// TwinCAT 3 PLC project PLC1
// ProgramVersion: 3.1.4026.21
// libraries:
//   Tc2_Standard, * (Beckhoff Automation GmbH)
//   Tc2_System, * (Beckhoff Automation GmbH)
//   Tc3_Module, * (Beckhoff Automation GmbH)
// project tree:
//   DUTs/ Jog_FxA_Type.TcDUT, Jog_FxB_Type.TcDUT, LaserJog.TcDUT, LaserVar.TcDUT, MyCustomType.TcDUT, SideClampVar.TcDUT
//   GVLs/ GVL.TcGVL, GVL_Main.TcGVL, Hmi_web.TcGVL
//   / PlcTask.TcTTO
//   POUs/ MAIN.TcPOU
// real-time tasks:
//   TASK PlcTask: cycle T#10ms, priority 20, ADS port 350

CONFIGURATION PLC1
    RESOURCE PLC ON TwinCAT3
        TASK PlcTask(INTERVAL := T#10ms, PRIORITY := 20);
        PROGRAM MAIN WITH PlcTask : MAIN;
    END_RESOURCE
END_CONFIGURATION

// ---- DUTs/Jog_FxA_Type.TcDUT
TYPE Jog_FxA_Type :
STRUCT
	
 H_Open:  BOOL;
 H_Open_S:  BOOL;
 H_Close:  BOOL;
 H_Close_S:  BOOL;

 H_Hold:  BOOL;
 H_Hold_S:  BOOL;

 V_Open:  BOOL;
 V_Open_S: BOOL;
 V_Close: BOOL;
 V_Close_S: BOOL;
  P : BOOL;
 P_S : BOOL;
 N : BOOL;
 N_S : BOOL;
 P_Fast : BOOL;
 P_Fast_S : BOOL;
 N_Fast : BOOL;
 N_Fast_S : BOOL;
END_STRUCT
END_TYPE

// ---- DUTs/Jog_FxB_Type.TcDUT
TYPE Jog_FxB_Type :
STRUCT
	 H_Open:  BOOL;
 H_Open_S:  BOOL;
 H_Close:  BOOL;
 H_Close_S:  BOOL;

 H_Hold:  BOOL;
 H_Hold_S:  BOOL;

 V_Open:  BOOL;
 V_Open_S: BOOL;
 V_Close: BOOL;
 V_Close_S: BOOL;

 
END_STRUCT
END_TYPE

// ---- DUTs/LaserJog.TcDUT
TYPE LaserJog :
STRUCT
	 X_P: BOOL;
     X_N: BOOL;
     X_H: BOOL;
	 
	 
	 X_P_S: BOOL;
     X_N_S: BOOL;
     X_H_S: BOOL;
	 
     Y_P: BOOL;
     Y_N: BOOL;
     Y_H: BOOL;
	 
	 
     Y_P_S: BOOL;
     Y_N_S: BOOL;
     Y_H_S: BOOL;
	 
     Z_P: BOOL;
     Z_N: BOOL;
     Z_H: BOOL;
	 
     Z_P_S: BOOL;
     Z_N_S: BOOL;
     Z_H_S: BOOL;
     Laser_Preview:BOOL;
     Laser_Preview_Select: INT	;
     Laser_Blow: BOOL;
     Laser_Cover: BOOL;

END_STRUCT
END_TYPE

// ---- DUTs/LaserVar.TcDUT
TYPE LaserVar :
STRUCT
    sv_bPLCHandShaking : BOOL;
    sv_bIPCHandShaking    : BOOL;
END_STRUCT
END_TYPE

// ---- DUTs/MyCustomType.TcDUT
TYPE MyCustomType :
STRUCT
    isActive : BOOL;
    speed    : REAL;
    counter  : INT;
END_STRUCT
END_TYPE

// ---- DUTs/SideClampVar.TcDUT
TYPE SideClampVar :
STRUCT
    sv_bButtonFwd: BOOL;
	sv_bButtonBwd: BOOL;
END_STRUCT
END_TYPE

// ---- GVLs/GVL.TcGVL
{attribute 'qualified_only'}
VAR_GLOBAL
END_VAR

// ---- GVLs/GVL_Main.TcGVL
{attribute 'qualified_only'}
VAR_GLOBAL
    g_bStart     : BOOL := FALSE;
    g_iCounter   : INT := 0;
    g_fSpeed     : REAL := 1.5;
    testBoolean     : BOOL := FALSE;
	
 g_machineStatus : MyCustomType := (
        isActive := FALSE,
        speed    := 0.0,
        counter  := 0
    );
	

LaserVars1:LaserVar := (
sv_bPLCHandShaking:= FALSE,
sv_bIPCHandShaking:= FALSE
    );
	LaserVars2:LaserVar := (
sv_bPLCHandShaking:= FALSE,
sv_bIPCHandShaking:= FALSE
    );
	LaserVars3:LaserVar := (
sv_bPLCHandShaking:= FALSE,
sv_bIPCHandShaking:= FALSE
    );
	LaserVars4:LaserVar := (
sv_bPLCHandShaking:= FALSE,
sv_bIPCHandShaking:= FALSE
    );

	
SideClampVars1:SideClampVar := (
sv_bButtonFwd:= FALSE,
sv_bButtonBwd:= FALSE);
	
SideClampVars2:SideClampVar := (
sv_bButtonFwd:= FALSE,
sv_bButtonBwd:= FALSE
 );
	
	

	
	
	
	
	
	
	
	
END_VAR

// ---- GVLs/Hmi_web.TcGVL
{attribute 'qualified_only'}
VAR_GLOBAL
    Jog_Speed: INT;
 Oil_Pump:BOOL;
Jog_FxA:Jog_FxA_Type:= (
      H_Open:= FALSE,
      H_Open_S:= FALSE,
      H_Close:= FALSE,
      H_Close_S:= FALSE,

      H_Hold:= FALSE,
      H_Hold_S:= FALSE,

      V_Open:= FALSE,
      V_Open_S:= FALSE,
      V_Close:= FALSE,
      V_Close_S:= FALSE,
   
     P:= FALSE,
      P_S:= FALSE,
      N:= FALSE,
      N_S:= FALSE,
      P_Fast:= FALSE,
      P_Fast_S:= FALSE,
      N_Fast:= FALSE,
      N_Fast_S:= FALSE
    );
 
 
Jog_FxB : Jog_FxB_Type := (
       H_Open:= FALSE,
      H_Open_S:= FALSE,
      H_Close:= FALSE,
      H_Close_S:= FALSE,

      H_Hold:= FALSE,
      H_Hold_S:= FALSE,

      V_Open:= FALSE,
      V_Open_S:= FALSE,
      V_Close:= FALSE,
      V_Close_S:= FALSE

    
);


 

//右軸
Jog_Ga: LaserJog:=( 
     X_P:= FALSE,
     X_N:= FALSE,
     X_H:= FALSE,
     Y_P:= FALSE,
     Y_N:= FALSE,
     Y_H:= FALSE,
     Z_P:= FALSE,
     Z_N:= FALSE,
     Z_H:= FALSE,
     Laser_Preview:=FALSE,
     Laser_Preview_Select:= 1,
     Laser_Blow:= FALSE,
     Laser_Cover:= FALSE);
//上軸
    Jog_Gb: LaserJog:=( 
     X_P:= FALSE,
     X_N:= FALSE,
     X_H:= FALSE,
     Y_P:= FALSE,
     Y_N:= FALSE,
     Y_H:= FALSE,
     Z_P:= FALSE,
     Z_N:= FALSE,
     Z_H:= FALSE,
     Laser_Preview:=FALSE,
     Laser_Preview_Select:= 1,
     Laser_Blow:= FALSE,
     Laser_Cover:= FALSE);
//左軸
    Jog_Gc: LaserJog:=( 
     X_P:= FALSE,
     X_N:= FALSE,
     X_H:= FALSE,
     Y_P:= FALSE,
     Y_N:= FALSE,
     Y_H:= FALSE,
     Z_P:= FALSE,
     Z_N:= FALSE,
     Z_H:= FALSE,
     Laser_Preview:=FALSE,
     Laser_Preview_Select:= 1,
     Laser_Blow:= FALSE,
     Laser_Cover:= FALSE);
//下軸
    Jog_Gd: LaserJog:=( 
     X_P:= FALSE,
     X_N:= FALSE,
     X_H:= FALSE,
     Y_P:= FALSE,
     Y_N:= FALSE,
     Y_H:= FALSE,
     Z_P:= FALSE,
     Z_N:= FALSE,
     Z_H:= FALSE,
     Laser_Preview:=FALSE,
     Laser_Preview_Select:= 1,
     Laser_Blow:= FALSE,
     Laser_Cover:= FALSE);


 	//*自動加工 */
    Auto_Start:  BOOL;
    //插單*/
    Auto_OneCycle_Start:  BOOL;
 	// 自動流程 加工單
	Auto_ProjectWorkOrder_uuid: STRING;
	// 排版專案 
    Start_WorkOrder_UUID: STRING;
	// 加工data_uuid
    Process_Data_UUID: STRING;
	// 雷標動作啟動 
    Process_Data_UUID_Start: BOOL;
 
 
 

    //動力滾輪
    Roller_Fwd:  BOOL;
    Roller_Fwd_S:  BOOL;
    //動力滾輪反轉
    Roller_Rev:  BOOL;
    Roller_Rev_S:  BOOL;

    //滾輪上浮
    Roller_Up:  BOOL;
    Roller_Up_S:  BOOL;
    //滾輪下降
    Roller_Down:  BOOL;
    Roller_Down_S:  BOOL;

    //入口料架-出口料架(0/1)*/
    Site_Select:  INT;
    //料架速率(0/1)*/
    Speed_Select:  INT;

    // 指定橫移->用二進位儲存 */
    Module_Select:  INT;

    //料架動作-台車前進*/
    Car_Rev:  BOOL;
    Car_Rev_S:  BOOL;
    //料架動作-台車後退
    Car_Fwd:  BOOL;
    Car_Fwd_S:  BOOL;
    //料架動作-台車上升
    Car_Up: BOOL;
    Car_Up_S:  BOOL;
    //料架動作-台車中間
    Car_Midd:  BOOL;
    Car_Midd_S:  BOOL;

    //料架動作-台車下降
    Car_Down:  BOOL;
    Car_Down_S:  BOOL;

    //料架動作-靠邊
    Pull_over_Push: BOOL;
    Pull_over_Push_S: BOOL;

    //料架動作-頂料柱上升
    StopPin_Up: BOOL;
    StopPin_Up_S:  BOOL;

    //料架動作-頂料柱下降
    StopPin_Down: BOOL;
    StopPin_Down_S: BOOL;

END_VAR

// ---- POUs/MAIN.TcPOU
PROGRAM MAIN
VAR
END_VAR

END_PROGRAM
